// TIA Portal V18 export
DATA_BLOCK "Xray_related_FB_DB"   // DB16
VERSION : 0.1
// stored: AutoNumber true, DBAccessibleFromOPCUA true, InstanceOfName Xray_related_FB, InstanceOfType FB
"Xray_related_FB"
   // VAR_OUTPUT
   //    fpd_power : Bool;
   // END_VAR
BEGIN
END_DATA_BLOCK
